Fanuc KAREL source: SET_POS_TPE.kl

PROGRAM T
%NOLOCKGROUP
VAR
 v0 : INTEGER
 v1 : INTEGER
 v2 : XYZWPR
 v3 : INTEGER
 v4 : INTEGER
BEGIN
 SET_POS_TPE(v0, v1, v2, v3, v4)
END T
